{attribute 'qualified_only'}
VAR_GLOBAL 
	TDKLoad : ARRAY [1..8] OF ST_Setpoints_Base;
	GLSLoad : ST_Setpoints_Base;
	GLS1_VSP : DINT := 50;
	GLS2_VSP : DINT := 50;
END_VAR

(* stored: Version 1.1.0.1, ProductVersion 3.1.4024.11
   GVL Setpoints: Id {5ed1e99e-ec63-45e6-b291-ebd24a0848f8} *)
